// TIA Portal V20 export
DATA_BLOCK "instLER_visionHistory"   // DB304
// stored: InstanceOfName LER_visionHistory, InstanceOfType FB
"LER_visionHistory"
   // VAR_INPUT
   //    trigger : Bool;
   //    result : "LER_typePartData";
   // END_VAR
   // VAR_IN_OUT
   //    dataHistory : "LER_typeVisionHistory";
   // END_VAR
   // VAR
   //    statDeleteData : "LER_typeVisionHistory";
   //    statTrigger : Array[0..99] of Bool;
   //    statTonTimer { S7_SetPoint := 'True'} : Array[0..99] of TON_TIME;
   //    statComplete : Array[0..99] of Bool;
   // END_VAR
BEGIN
END_DATA_BLOCK
